// TIA Portal project "项目工作" (V16)

(* hardware
DEVICE "S7-1200 station_1"  S7-1200 Station
   slot 0: "Rack_0"  S7-1200 Rack  Rack  V1.0
   slot 1: "项目工作平台"  CPU 1215C DC/DC/DC  6ES7 215-1AG40-0XB0  V4.2
   slot 2: "DI 16x24VDC/DQ 16xRelay_1"  SM 1223 DI16/DQ16 x relay  6ES7 223-1PL32-0XB0  V2.0
   slot 3: "DI 8x24VDC/DQ 8xRelay_1"  SM 1223 DI8/DQ8 x relay  6ES7 223-1PH32-0XB0  V2.0
   slot 4: "DI 16x24VDC_1"  6ES7 221-1BH32-0XB0  V2.0
DEVICE "GSD device_1"  GSD.Device.PN
   slot 0: "机架"  Rack  V1.0
   slot 0: "is2000"  In-Sight IS2XXX CC-B  IS2XXX  5.9.1
      slot 0: "In-Sight IS2XXX CC-B"  In-Sight IS2XXX CC-B  5.9.1
      slot 1: "接口"  Interface
         slot 1: "端口 1"  Port 1
   slot 1: "采集控制_1"  Acquisition Control  5.9.1
      slot 0: "采集控制"  Acquisition Control  5.9.1
   slot 2: "采集状态_1"  Acquisition Status  5.9.1
      slot 0: "采集状态"  Acquisition Status  5.9.1
   slot 3: "检查控件_1"  Inspection Control  5.9.1
      slot 0: "检查控件"  Inspection Control  5.9.1
   slot 4: "检查状态_1"  Inspection Status  5.9.1
      slot 0: "检查状态"  Inspection Status  5.9.1
   slot 5: "命令控制_1"  Command Control  5.9.1
      slot 0: "命令控制"  Command Control  5.9.1
   slot 6: "SoftEvent 控制_1"  SoftEvent Control  5.9.1
      slot 0: "SoftEvent 控制"  SoftEvent Control  5.9.1
   slot 7: "用户数据 - 64 个字节_1"  User Data - 64 bytes  5.9.1
      slot 0: "用户数据 - 64 个字节"  User Data - 64 bytes  5.9.1
   slot 8: "结果 - 64 个字节_1"  Results - 64 bytes  5.9.1
      slot 0: "结果 - 64 个字节"  Results - 64 bytes  5.9.1
*)

// ===== PLC "项目工作平台"  CPU 1215C DC/DC/DC =====

VAR_GLOBAL   // PLC tag table "默认变量表"
   "System_Byte" AT %MB1 : Byte;
   "FirstScan" AT %M1.0 : Bool;
   "DiagStatusUpdate" AT %M1.1 : Bool;
   "AlwaysTRUE" AT %M1.2 : Bool;
   "AlwaysFALSE" AT %M1.3 : Bool;
   "Clock_Byte" AT %MB0 : Byte;
   "Clock_10Hz" AT %M0.0 : Bool;
   "Clock_5Hz" AT %M0.1 : Bool;
   "Clock_2.5Hz" AT %M0.2 : Bool;
   "Clock_2Hz" AT %M0.3 : Bool;
   "Clock_1.25Hz" AT %M0.4 : Bool;
   "Clock_1Hz" AT %M0.5 : Bool;
   "Clock_0.625Hz" AT %M0.6 : Bool;
   "Clock_0.5Hz" AT %M0.7 : Bool;
END_VAR

VAR_GLOBAL   // PLC tag table "相机"
   "ii_ID1" AT %IW74 : Int;
   "ii_ID2" AT %IW76 : Int;
   "ii_N1_X" AT %ID80 : Real;
   "ii_N1_Y" AT %ID84 : Real;
   "ii_N1_A" AT %ID88 : Real;
   "ii_N2_X" AT %ID92 : Real;
   "ii_N2_Y" AT %ID96 : Real;
   "ii_N2_A" AT %ID100 : Real;
   "ii_N3_X" AT %ID104 : Real;
   "ii_N3_Y" AT %ID108 : Real;
   "ii_N3_A" AT %ID112 : Real;
   "ii_ID3" AT %IW78 : Int;
   "相机采集控制" AT %QB5 : Byte;
   "相机拍照完成" AT %I7.1 : Bool;
END_VAR

VAR_GLOBAL   // PLC tag table "IO输入"
   "光电门1" AT %I2.0 : Bool;
   "光电门2" AT %I2.1 : Bool;
   "抓取位光电门3" AT %I2.2 : Bool;
END_VAR

VAR_GLOBAL   // PLC tag table "IO输出"
   "拍照位气缸" AT %Q3.0 : Bool;
   "抓取位气缸" AT %Q3.1 : Bool;
   "交流电机正转" AT %Q2.4 : Bool;
END_VAR

DATA_BLOCK "相机流水线_DB"   // DB1
{ S7_Optimized_Access := 'TRUE' }
VERSION : 0.1
// stored: InstanceOfName 相机流水线
"相机流水线"
BEGIN
END_DATA_BLOCK

DATA_BLOCK "数据块_1"   // DB2
{ S7_Optimized_Access := 'TRUE' }
VERSION : 0.1
BEGIN
END_DATA_BLOCK

// folder: System blocks/Program resources

DATA_BLOCK "IEC_Timer_0_DB"   // DB3
{ S7_Optimized_Access := 'TRUE' }
AUTHOR : Simatic
FAMILY : IEC
NAME : IEC_TMR
VERSION : 1.0
// stored: InstanceOfName IEC_TIMER
"IEC_TIMER"
BEGIN
END_DATA_BLOCK

DATA_BLOCK "IEC_Timer_0_DB_1"   // DB4
{ S7_Optimized_Access := 'TRUE' }
AUTHOR : Simatic
FAMILY : IEC
NAME : IEC_TMR
VERSION : 1.0
// stored: InstanceOfName IEC_TIMER
"IEC_TIMER"
BEGIN
END_DATA_BLOCK

DATA_BLOCK "IEC_Timer_0_DB_2"   // DB5
{ S7_Optimized_Access := 'TRUE' }
AUTHOR : Simatic
FAMILY : IEC
NAME : IEC_TMR
VERSION : 1.0
// stored: InstanceOfName IEC_TIMER
"IEC_TIMER"
BEGIN
END_DATA_BLOCK

DATA_BLOCK "IEC_Timer_0_DB_3"   // DB6
{ S7_Optimized_Access := 'TRUE' }
AUTHOR : Simatic
FAMILY : IEC
NAME : IEC_TMR
VERSION : 1.0
// stored: InstanceOfName IEC_TIMER
"IEC_TIMER"
BEGIN
END_DATA_BLOCK

DATA_BLOCK "IEC_Timer_0_DB_4"   // DB7
{ S7_Optimized_Access := 'TRUE' }
AUTHOR : Simatic
FAMILY : IEC
NAME : IEC_TMR
VERSION : 1.0
// stored: InstanceOfName IEC_TIMER
"IEC_TIMER"
BEGIN
END_DATA_BLOCK

// folder: (top level)

FUNCTION_BLOCK "相机流水线"   // FB1, LAD
{ S7_Optimized_Access := 'TRUE' }
VERSION : 0.1
   VAR
      Ptrig : Struct
         "1" : Bool;
         "2" : Bool;
         "3" : Bool;
      END_STRUCT;
      相机 : Struct
         拍照 : Bool;
      END_STRUCT;
      交流电机 : Struct
         正转 : Bool;
         停止 : Bool;
      END_STRUCT;
   END_VAR
   VAR_TEMP
      "1" : Bool;
      "2" : Bool;
   END_VAR
   VAR_TEMP   // added for the SCL form of the ladder/FBD networks
      _w1 : Bool;
      _w2 : Bool;
   END_VAR
BEGIN

REGION Network 1
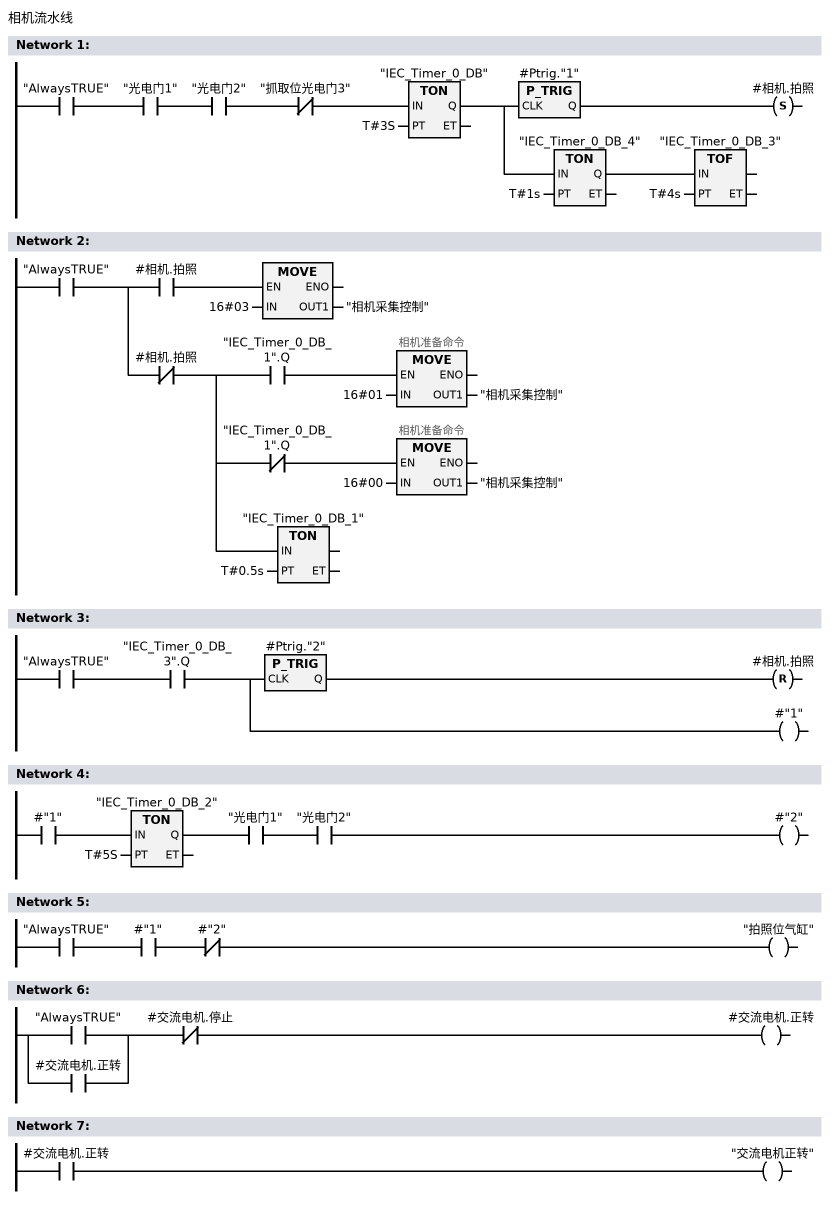
   "IEC_Timer_0_DB".TON(IN := "AlwaysTRUE" AND "光电门1" AND "光电门2" AND NOT "抓取位光电门3", PT := T#3S);
   #_w1 := "IEC_Timer_0_DB".Q AND NOT #Ptrig."1";   // rising edge
   #Ptrig."1" := "IEC_Timer_0_DB".Q;
   IF #_w1 THEN #相机.拍照 := TRUE; END_IF;
   "IEC_Timer_0_DB_4".TON(IN := "IEC_Timer_0_DB".Q, PT := T#1s);
   "IEC_Timer_0_DB_3".TOF(IN := "IEC_Timer_0_DB_4".Q, PT := T#4s);
END_REGION

REGION Network 2
   IF "AlwaysTRUE" AND #相机.拍照 THEN "相机采集控制" := 16#03; END_IF;
   #_w1 := "AlwaysTRUE" AND NOT #相机.拍照;
   IF #_w1 AND "IEC_Timer_0_DB_1".Q THEN
       "相机采集控制" := 16#01;   // 相机准备命令
   END_IF;
   IF #_w1 AND NOT "IEC_Timer_0_DB_1".Q THEN
       "相机采集控制" := 16#00;   // 相机准备命令
   END_IF;
   "IEC_Timer_0_DB_1".TON(IN := #_w1, PT := T#0.5s);
END_REGION

REGION Network 3
   RUNG wire#powerrail
      Contact( "AlwaysTRUE" )
      Contact( "IEC_Timer_0_DB_3".Q )
      wire#w1
      P_Trig( #Ptrig."2" )
      R_Coil( #相机.拍照 )
   END_RUNG
   RUNG wire#w1
      Coil( #"1" )
   END_RUNG
   // the same network as SCL:
   #_w1 := "AlwaysTRUE" AND "IEC_Timer_0_DB_3".Q;
   #_w2 := #_w1 AND NOT #Ptrig."2";   // rising edge
   #Ptrig."2" := #_w1;
   IF #_w2 THEN #相机.拍照 := FALSE; END_IF;
   #"1" := #_w1;
END_REGION

REGION Network 4
   "IEC_Timer_0_DB_2".TON(IN := #"1", PT := T#5S);
   #"2" := "IEC_Timer_0_DB_2".Q AND "光电门1" AND "光电门2";
END_REGION

REGION Network 5
   RUNG wire#powerrail
      Contact( "AlwaysTRUE" )
      Contact( #"1" )
      I_Contact( #"2" )
      Coil( "拍照位气缸" )
   END_RUNG
   // the same network as SCL:
   "拍照位气缸" := "AlwaysTRUE" AND #"1" AND NOT #"2";
END_REGION

REGION Network 6
   RUNG wire#powerrail
      Contact( "AlwaysTRUE" )
      wire#w1
      I_Contact( #交流电机.停止 )
      Coil( #交流电机.正转 )
   END_RUNG
   RUNG wire#powerrail
      Contact( #交流电机.正转 )
   END_RUNG wire#w1
   // the same network as SCL:
   #交流电机.正转 := ("AlwaysTRUE" OR #交流电机.正转) AND NOT #交流电机.停止;
END_REGION

REGION Network 7
   RUNG wire#powerrail
      Contact( #交流电机.正转 )
      Coil( "交流电机正转" )
   END_RUNG
   // the same network as SCL:
   "交流电机正转" := #交流电机.正转;
END_REGION

REGION Network 8 (SCL)
   (* /*
       1：直径60，高度40；颜色black；
       2：高45，直径35；颜色red；
       //3：高11，直径35，颜色blue；
       4；高28，直径60，颜色黑色；

       标定x1=210，x2=292，像数值82，实际值245，
       82/245=0.3346938775510204；
       245/82=2.98780487804878；



       New：
       1：201 482
       //60/281=0.2135
       60/268=0.2238
       2：264 426
       35/156=0.2243
       3：230 500
       60/254=0.2362
   */ *)
   //机器人抓取好工件，发送信号过来，然后数组 GVL".相机.数据组 移动，
END_REGION
END_FUNCTION_BLOCK

ORGANIZATION_BLOCK "Main"   // OB1, LAD, ProgramCycle
TITLE = "Main Program Sweep (Cycle)"
{ S7_Optimized_Access := 'TRUE' }
VERSION : 0.1
   VAR_INPUT
      Initial_Call : Bool;   // Initial call of this OB
      Remanence : Bool;   // =True, if remanent data are available
   END_VAR
BEGIN

REGION Network 1
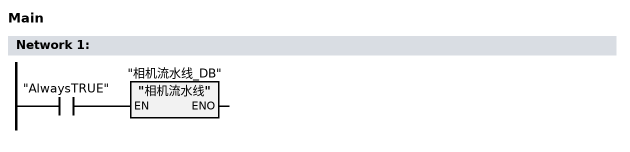
   RUNG wire#powerrail
      Contact( "AlwaysTRUE" )
      "相机流水线_DB"()
   END_RUNG
   // the same network as SCL:
   IF "AlwaysTRUE" THEN
       "相机流水线_DB"();   // "相机流水线"
   END_IF;
END_REGION
END_ORGANIZATION_BLOCK